Yaskawa INFORM job: TGGGGVF.JBI

/JOB
//NAME TGGGGVF
//POS
///NPOS 0,0,0,0,0,0
//INST
///DATE 2023/12/14 17:07
///ATTR SC,RW,RJ
////FRAME ROBOT
///GROUP1 RB1,BS1
NOP
END
